// TIA Portal V17 export
// export: Created 2024-08-09T12:53:11.5951198Z, ExportSetting WithDefaults, DisplayName Totally Integrated Automation Portal, DisplayVersion V17 Update 7, DisplayName TIA Portal Openness, DisplayVersion V17 Update 7, DisplayName TIA Portal Version Control Interface, DisplayVersion V17, DisplayName STEP 7 Professional, DisplayVersion V17 Update 7, DisplayName STEP 7 Safety, DisplayVersion V17 Update 6, DisplayName WinCC Professional, DisplayVersion V17 Update 7
VAR_GLOBAL   // PLC tag table "Dosage_Gen"
END_VAR
VAR_GLOBAL CONSTANT   // user constants
   NB_MAX_LIQ_MEL : USInt := 10;
   NB_MAX_BR : USInt := 1;
   NB_CIR_EXP : USInt := 9;
END_VAR
